    rq_wait_ft_sensor_steady(2000)
    zero_ftsensor()
    sleep(0.1)
    # end: URCap Program Node
    # begin: URCap Program Node
    #   Source: Robotiq_Copilot, 1.22.1.14215, Robotiq Inc.
    #   Type: Find Surface
    $ 88 "Find Surface"
    zero_ftsensor()
    sleep(0.1)
    surface_found = rq_linear_search_urcap("Z+", 10.000, 0.005000, 0.100000, 1)
    storevar.setvariablepose("rq_findSurface_ef5e6fd5-1d3d-43c2-9922-b9c2fd55821a_exitPosition", get_actual_tcp_pose())
    $ 89 "'Add Stop conditions from the Find Surface node'" "noBreak"
    # 'Add Stop conditions from the Find Surface node'
    # end: URCap Program Node
    # begin: URCap Program Node
    #   Source: Robotiq_Copilot, 1.22.1.14215, Robotiq Inc.
    #   Type: Finishing Tool Control
    $ 90 "Start tool"
    set_standard_digital_out(0, True)
    # end: URCap Program Node
    $ 91 "Wait: 0.5"
    sleep(0.5)
    $ 92 "Force"
    sleep(0.02)
    zero_ftsensor()
    force_mode(tool_pose(), [0, 0, 1, 0, 0, 0], [0.0, 0.0, 5.0, 0.0, 0.0, 0.0], 2, [0.1, 0.1, 0.15, 0.3490658503988659, 0.3490658503988659, 0.3490658503988659])
    $ 93 "Waypoint_7" "noBreak"
    set_tcp(p[0.00318,0.11464,0.09820000000000001,-0.7853981633974483,0.0,0.0])
    movel(pose_trans(CubeFront, pose_trans(p[.002249871974, -.169402369556, .608081756259, .020435046430, 2.223511403835, 2.209446612627], Waypoint_7_p)), a=1.2, v=0.05)
    end_force_mode()
    stopl(5.0)
    # begin: URCap Program Node
    #   Source: Robotiq_Copilot, 1.22.1.14215, Robotiq Inc.
    #   Type: Finishing Tool Control
    $ 94 "Stop tool"
    set_standard_digital_out(0, False)
    # end: URCap Program Node
    $ 95 "Waypoint_13" "breakAfter"
    set_tcp(p[0.00318,0.11464,0.09820000000000001,-0.7853981633974483,0.0,0.0])
    movel(pose_trans(CubeFront, pose_trans(p[-.002001169423, -.178123008725, .618090231485, -1.568699287997, .013964727372, .007428573496], Waypoint_13_p)), a=1.2, v=0.25)
    $ 96 "Waypoint_9" "breakAfter"
    set_tcp(p[0.00318,0.11464,0.09820000000000001,-0.7853981633974483,0.0,0.0])
    movel(pose_trans(CubeFront, pose_trans(p[-.002001169423, -.178123008725, .618090231485, -1.568699287997, .013964727372, .007428573496], Waypoint_9_p)), a=1.2, v=0.25)
    $ 97 "Clear" "breakAfter"
    set_tcp(p[0.00318,0.11464,0.09820000000000001,-0.7853981633974483,0.0,0.0])
    movel(pose_trans(CubeFront, pose_trans(p[.002249871974, -.169402369556, .608081756259, .020435046430, 2.223511403835, 2.209446612627], Clear_p)), a=1.2, v=0.25)
  end
  def SprayFront():
    $ 98 "SprayFront" "noBreak"
    $ 99 "SprayFront"
    $ 100 "MoveJ"
    $ 101 "SprayClear" "breakAfter"
    set_tcp(p[0.020839023181949995,-0.027139950822234082,0.10599373590389219,0.12258870209179472,1.1769383890382668,2.869747076630172])
    movej(get_inverse_kin(pose_trans(SprayPlane, pose_trans(p[.380158499114, -.183027591855, .571104219868, -1.574901506950, .032921162495, .010611987369], SprayClear_p)), qnear=SprayClear_q), a=1.3962634015954636, v=1.0471975511965976)
    $ 102 "MoveJ"
    $ 103 "Waypoint_10" "breakAfter"
    set_tcp(p[0.020839023181949995,-0.027139950822234082,0.10599373590389219,0.12258870209179472,1.1769383890382668,2.869747076630172])
    movej(get_inverse_kin(pose_trans(SprayPlane, pose_trans(p[.380158499114, -.183027591855, .571104219868, -1.574901506950, .032921162495, .010611987369], Waypoint_10_p)), qnear=Waypoint_10_q), a=1.3962634015954636, v=1.0471975511965976)
    $ 104 "Set DO[1]=On"
    set_standard_digital_out(1, True)
    $ 105 "MoveL"
    $ 106 "Waypoint_12" "breakAfter"
    movel(pose_trans(SprayPlane, pose_trans(p[.380158499114, -.183027591855, .571104219868, -1.574901506950, .032921162495, .010611987369], Waypoint_12_p)), a=1.2, v=0.1)
    $ 107 "Set DO[1]=Off"
    set_standard_digital_out(1, False)
    $ 108 "MoveJ"
    $ 109 "Waypoint_21" "breakAfter"
    set_tcp(p[0.020839023181949995,-0.027139950822234082,0.10599373590389219,0.12258870209179472,1.1769383890382668,2.869747076630172])
    movej(get_inverse_kin(pose_trans(SprayPlane, pose_trans(p[.380158499114, -.183027591855, .571104219868, -1.574901506950, .032921162495, .010611987369], Waypoint_21_p)), qnear=Waypoint_21_q), a=1.3962634015954636, v=1.0471975511965976)
    $ 110 "Set DO[1]=On"
    set_standard_digital_out(1, True)
    $ 111 "MoveL"
    $ 112 "Waypoint_22" "breakAfter"
    set_tcp(p[0.020839023181949995,-0.027139950822234082,0.10599373590389219,0.12258870209179472,1.1769383890382668,2.869747076630172])
    movel(pose_trans(SprayPlane, pose_trans(p[.380158499114, -.183027591855, .571104219868, -1.574901506950, .032921162495, .010611987369], Waypoint_22_p)), a=1.2, v=0.1)
    $ 113 "Set DO[1]=Off"
    set_standard_digital_out(1, False)
    $ 114 "MoveJ"
    $ 115 "Waypoint_23" "breakAfter"
    set_tcp(p[0.020839023181949995,-0.027139950822234082,0.10599373590389219,0.12258870209179472,1.1769383890382668,2.869747076630172])
    movej(get_inverse_kin(pose_trans(SprayPlane, pose_trans(p[.380158499114, -.183027591855, .571104219868, -1.574901506950, .032921162495, .010611987369], Waypoint_23_p)), qnear=Waypoint_23_q), a=1.3962634015954636, v=1.0471975511965976)
    $ 116 "Set DO[1]=On"
    set_standard_digital_out(1, True)
    $ 117 "MoveL"
    $ 118 "Waypoint_24" "breakAfter"
    set_tcp(p[0.020839023181949995,-0.027139950822234082,0.10599373590389219,0.12258870209179472,1.1769383890382668,2.869747076630172])
    movel(pose_trans(SprayPlane, pose_trans(p[.380158499114, -.183027591855, .571104219868, -1.574901506950, .032921162495, .010611987369], Waypoint_24_p)), a=1.2, v=0.1)
    $ 119 "Set DO[1]=Off"
    set_standard_digital_out(1, False)
    $ 120 "MoveJ"
    $ 121 "Waypoint_38" "breakAfter"
    set_tcp(p[0.020839023181949995,-0.027139950822234082,0.10599373590389219,0.12258870209179472,1.1769383890382668,2.869747076630172])
    movej(get_inverse_kin(pose_trans(SprayPlane, pose_trans(p[.152076837040, -.186455621862, .570552501782, -1.567181840228, .028822735400, .008142754325], Waypoint_38_p)), qnear=Waypoint_38_q), a=1.3962634015954636, v=1.0471975511965976)
    $ 122 "Set DO[1]=On"
    set_standard_digital_out(1, True)
    $ 123 "MoveL"
    $ 124 "Waypoint_25" "breakAfter"
    set_tcp(p[0.020839023181949995,-0.027139950822234082,0.10599373590389219,0.12258870209179472,1.1769383890382668,2.869747076630172])
    movel(pose_trans(SprayPlane, pose_trans(p[.380158499114, -.183027591855, .571104219868, -1.574901506950, .032921162495, .010611987369], Waypoint_25_p)), a=1.2, v=0.1)
    $ 125 "Set DO[1]=Off"
    set_standard_digital_out(1, False)
    $ 126 "MoveJ"
    $ 127 "SprayClear" "breakAfter"
    set_tcp(p[0.020839023181949995,-0.027139950822234082,0.10599373590389219,0.12258870209179472,1.1769383890382668,2.869747076630172])
    movej(get_inverse_kin(pose_trans(SprayPlane, pose_trans(p[.380158499114, -.183027591855, .571104219868, -1.574901506950, .032921162495, .010611987369], SprayClear_p)), qnear=SprayClear_q), a=1.3962634015954636, v=1.0471975511965976)
  end
  def SprayRebate():
    $ 128 "SprayRebate" "noBreak"
    $ 129 "SprayRebate"
    $ 130 "MoveJ"
    $ 131 "SprayClear" "breakAfter"
    set_tcp(p[0.020839023181949995,-0.027139950822234082,0.10599373590389219,0.12258870209179472,1.1769383890382668,2.869747076630172])
    movej(get_inverse_kin(pose_trans(SprayPlane, pose_trans(p[.380158499114, -.183027591855, .571104219868, -1.574901506950, .032921162495, .010611987369], SprayClear_p)), qnear=SprayClear_q), a=1.3962634015954636, v=1.0471975511965976)
    $ 132 "MoveJ"
    $ 133 "Waypoint_28" "breakAfter"
    set_tcp(p[0.020839023181949995,-0.027139950822234082,0.10599373590389219,0.12258870209179472,1.1769383890382668,2.869747076630172])
    movej(get_inverse_kin(pose_trans(SprayPlane, pose_trans(p[-.002001169423, -.178123008725, .618090231485, -1.568699287997, .013964727372, .007428573496], Waypoint_28_p)), qnear=Waypoint_28_q), a=1.3962634015954636, v=1.0471975511965976)
    $ 134 "Set DO[1]=On"
    set_standard_digital_out(1, True)
    $ 135 "MoveL"
    $ 136 "Waypoint_27" "breakAfter"
    set_tcp(p[0.020839023181949995,-0.027139950822234082,0.10599373590389219,0.12258870209179472,1.1769383890382668,2.869747076630172])
    movel(pose_trans(SprayPlane, pose_trans(p[-.002001169423, -.178123008725, .618090231485, -1.568699287997, .013964727372, .007428573496], Waypoint_27_p)), a=1.2, v=0.1)
    $ 137 "Set DO[1]=Off"
    set_standard_digital_out(1, False)
    $ 138 "MoveJ"
    $ 139 "Waypoint_29" "breakAfter"
    set_tcp(p[0.020839023181949995,-0.027139950822234082,0.10599373590389219,0.12258870209179472,1.1769383890382668,2.869747076630172])
    movej(get_inverse_kin(pose_trans(SprayPlane, pose_trans(p[-.002001169423, -.178123008725, .618090231485, -1.568699287997, .013964727372, .007428573496], Waypoint_29_p)), qnear=Waypoint_29_q), a=1.3962634015954636, v=1.0471975511965976)
    $ 140 "Set DO[1]=On"
    set_standard_digital_out(1, True)
    $ 141 "MoveL"
    $ 142 "Waypoint_30" "breakAfter"
    set_tcp(p[0.020839023181949995,-0.027139950822234082,0.10599373590389219,0.12258870209179472,1.1769383890382668,2.869747076630172])
    movel(pose_trans(SprayPlane, pose_trans(p[-.002001169423, -.178123008725, .618090231485, -1.568699287997, .013964727372, .007428573496], Waypoint_30_p)), a=1.2, v=0.1)
    $ 143 "Set DO[1]=Off"
    set_standard_digital_out(1, False)
    $ 144 "MoveJ"
    $ 145 "SprayClear" "breakAfter"
    set_tcp(p[0.020839023181949995,-0.027139950822234082,0.10599373590389219,0.12258870209179472,1.1769383890382668,2.869747076630172])
    movej(get_inverse_kin(pose_trans(SprayPlane, pose_trans(p[.380158499114, -.183027591855, .571104219868, -1.574901506950, .032921162495, .010611987369], SprayClear_p)), qnear=SprayClear_q), a=1.3962634015954636, v=1.0471975511965976)
    $ 146 "MoveJ"
    $ 147 "Waypoint_32" "breakAfter"
    set_tcp(p[0.020839023181949995,-0.027139950822234082,0.10599373590389219,0.12258870209179472,1.1769383890382668,2.869747076630172])
    movej(get_inverse_kin(pose_trans(SprayPlane, pose_trans(p[-.002001169423, -.178123008725, .618090231485, -1.568699287997, .013964727372, .007428573496], Waypoint_32_p)), qnear=Waypoint_32_q), a=1.3962634015954636, v=1.0471975511965976)
    $ 148 "Set DO[1]=On"
    set_standard_digital_out(1, True)
    $ 149 "MoveL"
    $ 150 "Waypoint_33" "breakAfter"
    set_tcp(p[0.020839023181949995,-0.027139950822234082,0.10599373590389219,0.12258870209179472,1.1769383890382668,2.869747076630172])
    movel(pose_trans(SprayPlane, pose_trans(p[-.002001169423, -.178123008725, .618090231485, -1.568699287997, .013964727372, .007428573496], Waypoint_33_p)), a=1.2, v=0.1)
    $ 151 "Set DO[1]=Off"
    set_standard_digital_out(1, False)
    $ 152 "MoveJ"
    $ 153 "SprayClear" "breakAfter"
    set_tcp(p[0.020839023181949995,-0.027139950822234082,0.10599373590389219,0.12258870209179472,1.1769383890382668,2.869747076630172])
    movej(get_inverse_kin(pose_trans(SprayPlane, pose_trans(p[.380158499114, -.183027591855, .571104219868, -1.574901506950, .032921162495, .010611987369], SprayClear_p)), qnear=SprayClear_q), a=1.3962634015954636, v=1.0471975511965976)
  end
  def SandFront():
    $ 154 "SandFront" "noBreak"
    $ 155 "sandFront"
    $ 156 "MoveJ"
    $ 157 "Waypoint_35" "breakAfter"
    set_tcp(p[0.00318,0.11464,0.09820000000000001,-0.7853981633974483,0.0,0.0])
    movej(get_inverse_kin(pose_trans(Work, pose_trans(p[.002249871974, -.169402369556, .608081756259, .020435046430, 2.223511403835, 2.209446612627], Waypoint_35_p)), qnear=Waypoint_35_q), a=1.3962634015954636, v=1.0471975511965976)
    $ 158 "MoveL"
    $ 159 "Waypoint_1" "breakAfter"
    set_tcp(p[0.00318,0.11464,0.09820000000000001,-0.7853981633974483,0.0,0.0])
    movel(pose_trans(Work, pose_trans(p[-.005597006121, -.192408094989, .653246871754, -1.571622694982, -.002967386491, .002471774867], Waypoint_1_p)), a=1.2, v=0.25)
    # begin: URCap Program Node
    #   Source: Robotiq_Copilot, 1.22.1.14215, Robotiq Inc.
    #   Type: Zero FT Sensor
    $ 160 "Zero FT Sensor"

    rq_wait_ft_sensor_steady(2000)
    zero_ftsensor()
    sleep(0.1)
    # end: URCap Program Node
    # begin: URCap Program Node
    #   Source: Robotiq_Copilot, 1.22.1.14215, Robotiq Inc.
    #   Type: Find Surface
    $ 161 "Find Surface"
    surface_found = rq_linear_search_urcap("Z+", 10.000, 0.005000, 0.100000, 1)
    storevar.setvariablepose("rq_findSurface_7eeff1a3-6c12-4ed4-8857-ddcfb00799c6_exitPosition", get_actual_tcp_pose())
    $ 162 "'Add Stop conditions from the Find Surface node'" "noBreak"
    # 'Add Stop conditions from the Find Surface node'
    # end: URCap Program Node
    # begin: URCap Program Node
    #   Source: Robotiq_Copilot, 1.22.1.14215, Robotiq Inc.
    #   Type: Finishing Tool Control
    $ 163 "Start tool"
    set_standard_digital_out(0, True)
    # end: URCap Program Node
    $ 164 "Wait: 0.5"
    sleep(0.5)
    $ 165 "MoveL"
    $ 166 "Force"
    sleep(0.02)
    zero_ftsensor()
    force_mode(tool_pose(), [0, 0, 1, 0, 0, 0], [0.0, 0.0, 5.0, 0.0, 0.0, 0.0], 2, [0.1, 0.1, 0.15, 0.3490658503988659, 0.3490658503988659, 0.3490658503988659])
    $ 167 "Waypoint_34" "noBreak"
    set_tcp(p[0.00318,0.11464,0.09820000000000001,-0.7853981633974483,0.0,0.0])
    movel(pose_trans(Work, pose_trans(p[.002249871974, -.169402369556, .608081756259, .020435046430, 2.223511403835, 2.209446612627], Waypoint_34_p)), a=1.2, v=0.06)
    $ 168 "Waypoint_37" "noBreak"
    set_tcp(p[0.00318,0.11464,0.09820000000000001,-0.7853981633974483,0.0,0.0])
    movel(pose_trans(Work, pose_trans(p[.002249871974, -.169402369556, .608081756259, .020435046430, 2.223511403835, 2.209446612627], Waypoint_37_p)), a=1.2, v=0.06)
    $ 169 "Waypoint_36" "noBreak"
    set_tcp(p[0.00318,0.11464,0.09820000000000001,-0.7853981633974483,0.0,0.0])
    movel(pose_trans(Work, pose_trans(p[.002249871974, -.169402369556, .608081756259, .020435046430, 2.223511403835, 2.209446612627], Waypoint_36_p)), a=1.2, v=0.06)
    $ 170 "Waypoint_1" "noBreak"
    set_tcp(p[0.00318,0.11464,0.09820000000000001,-0.7853981633974483,0.0,0.0])
    movel(pose_trans(Work, pose_trans(p[-.005597006121, -.192408094989, .653246871754, -1.571622694982, -.002967386491, .002471774867], Waypoint_1_p)), a=1.2, v=0.06)
    # begin: URCap Program Node
    #   Source: Robotiq_Copilot, 1.22.1.14215, Robotiq Inc.
    #   Type: Finishing Tool Control
    $ 171 "Stop tool" "noBreak"
    set_standard_digital_out(0, False)
    # end: URCap Program Node
    end_force_mode()
    stopl(5.0)
    $ 172 "Direction: Tool Z-"
    global move_thread_flag_172=0
    thread move_thread_172():
      enter_critical
      move_thread_flag_172 = 1
      local towardsPos=calculate_point_to_move_towards(get_forward_kin(), [0.0,0.0,-1.0], 0.025)
      movel(towardsPos, a=1.2, v=0.06)
      move_thread_flag_172 = 2
      exit_critical
    end
    move_thread_flag_172 = 0
    move_thread_han_172 = run move_thread_172()
    while (True):
      sleep(1.0E-10)
      if (move_thread_flag_172 > 1):
        join move_thread_han_172
        $ 173 "Until (distance)"
        break
      end
      sync()
    end
    $ 174 "MoveJ"
    $ 175 "Waypoint_35" "breakAfter"
    movej(get_inverse_kin(pose_trans(Work, pose_trans(p[.002249871974, -.169402369556, .608081756259, .020435046430, 2.223511403835, 2.209446612627], Waypoint_35_p)), qnear=Waypoint_35_q), a=1.3962634015954636, v=1.0471975511965976)
  end
  def StartSpray():
    $ 176 "StartSpray" "noBreak"
    $ 177 "Set DO[1]=On"
    set_standard_digital_out(1, True)
    $ 178 "Wait: 0.3"
    sleep(0.3)
  end
  def stopSpray():
    $ 179 "stopSpray" "noBreak"
    $ 180 "Set DO[1]=Off"
    set_standard_digital_out(1, False)
    $ 181 "Wait: 0.3"
    sleep(0.3)
  end
  thread EventThread():
    while (True):
      if (get_standard_digital_in(1) !=   True  ):
        $ 49 "Set DO[0]=Off"
        set_standard_digital_out(0, False)
        $ 50 "Set DO[1]=Off"
        set_standard_digital_out(1, False)
        $ 51 "Halt"
        halt
      end
      sync()
    end
  end
  eventThread = run EventThread()
  $ 1 "Robot Program"
  $ 2 "Main"
  $ 3 "MoveJ"
  $ 4 "Clear" "breakAfter"
  set_tcp(p[0.00318,0.11464,0.09820000000000001,-0.7853981633974483,0.0,0.0])
  movej(get_inverse_kin(pose_trans(CubeFront, pose_trans(p[.002249871974, -.169402369556, .608081756259, .020435046430, 2.223511403835, 2.209446612627], Clear_p)), qnear=Clear_q), a=1.3962634015954636, v=1.0471975511965976)
  # begin: URCap Program Node
  #   Source: Robotiq_Copilot, 1.22.1.14215, Robotiq Inc.
  #   Type: Zero FT Sensor
  $ 5 "Zero FT Sensor"

  rq_wait_ft_sensor_steady(2000)
  zero_ftsensor()
  sleep(0.1)
  # end: URCap Program Node
  $ 6 "Work≔CubeFront"
  global Work=CubeFront
  $ 7 "Call SandFront"
  SandFront()
  $ 8 "Call SandRebate"
  SandRebate()
  $ 9 "Work≔SandBack"
  global Work=SandBack
  $ 10 "Call SandFront"
  SandFront()
  $ 11 "MoveJ"
  $ 12 "SprayClear" "breakAfter"
  set_tcp(p[0.020839023181949995,-0.027139950822234082,0.10599373590389219,0.12258870209179472,1.1769383890382668,2.869747076630172])
  movej(get_inverse_kin(pose_trans(SprayPlane, pose_trans(p[.380158499114, -.183027591855, .571104219868, -1.574901506950, .032921162495, .010611987369], SprayClear_p)), qnear=SprayClear_q), a=1.3962634015954636, v=1.0471975511965976)
  # begin: URCap Program Node
  #   Source: Robotiq_Copilot, 1.22.1.14215, Robotiq Inc.
  #   Type: Zero FT Sensor
  $ 13 "Zero FT Sensor"

  rq_wait_ft_sensor_steady(2000)
  zero_ftsensor()
  sleep(0.1)
  # end: URCap Program Node
  $ 14 "Call SprayFront"
  SprayFront()
  $ 15 "Call SprayRebate"
  SprayRebate()
end
